{attribute 'qualified_only'}
{attribute 'strict'}
TYPE EmotorStatus :
(
	start := 0,
	running := 1,
	stopped := 2
);
END_TYPE

(* stored: Version 1.1.0.1, ProductVersion 3.1.4024.12
   DUT EmotorStatus: Id {84a447f1-dacb-4f0e-a00a-2ea62652beb0} *)
